(* PLC project Unnamed, Unknown Unnamed 1 *)
(* stored: creationDateTime 2025-07-25T06:08:21, modificationDateTime 2025-07-25T06:08:21 *)

CONFIGURATION Config0
  RESOURCE Res0 ON PLC
  END_RESOURCE
END_CONFIGURATION
